(* IEC 61131-3 sources: AXOpen/src/components.keyence.vision/ctrl/src/Axo_IV3 (part 2) *)

                IF inParent = NULL THEN
                    Messenger.Activate(UINT#1500,eAxoMessageCategory#Error);
                    Status.Error.Id := UINT#1500;
                    RETURN;
                END_IF;
                IF Config.HWIDs.HW_Device  = UINT#0 THEN
                    Messenger.Activate(UINT#1501,eAxoMessageCategory#Error);
                    Status.Error.Id := UINT#1501;
                    RETURN;
                END_IF;
                IF Config.HWIDs.HwID_CommandControl  = UINT#0 THEN
                    Messenger.Activate(UINT#1502,eAxoMessageCategory#Error);
                    Status.Error.Id := UINT#1502;
                    RETURN;
                END_IF;
                IF Config.HWIDs.HwID_CommandStatusBits  = UINT#0 THEN
                    Messenger.Activate(UINT#1503,eAxoMessageCategory#Error);
                    Status.Error.Id := UINT#1503;
                    RETURN;
                END_IF;
                IF Config.HWIDs.HwID_DeviceResultBits_1  = UINT#0 THEN
                    Messenger.Activate(UINT#1504,eAxoMessageCategory#Error);
                    Status.Error.Id := UINT#1504;
                    RETURN;
                END_IF;
                IF Config.HWIDs.HwID_DeviceStatusWords  = UINT#0 THEN
                    Messenger.Activate(UINT#1505,eAxoMessageCategory#Error);
                    Status.Error.Id := UINT#1505;
                    RETURN;
                END_IF;
                IF Config.HWIDs.HwID_DeviceStatistics  = UINT#0 THEN
                    Messenger.Activate(UINT#1506,eAxoMessageCategory#Error);
                    Status.Error.Id := UINT#1506;
                    RETURN;
                END_IF;
                IF Config.HWIDs.HwID_PositionAdjustResult  = UINT#0 THEN
                    Messenger.Activate(UINT#1507,eAxoMessageCategory#Error);
                    Status.Error.Id := UINT#1507;
                    RETURN;
                END_IF;
                IF Config.HWIDs.HwID_ToolResult_1  = UINT#0 THEN
                    Messenger.Activate(UINT#1508,eAxoMessageCategory#Error);
                    Status.Error.Id := UINT#1508;
                    RETURN;
                END_IF;
                IF Config.HWIDs.HwID_ToolResult_2  = UINT#0 THEN
                    Messenger.Activate(UINT#1509,eAxoMessageCategory#Error);
                    Status.Error.Id := UINT#1509;
                    RETURN;
                END_IF;
                IF Config.HWIDs.HwID_ToolResult_3  = UINT#0 THEN
                    Messenger.Activate(UINT#1510,eAxoMessageCategory#Error);
                    Status.Error.Id := UINT#1510;
                    RETURN;
                END_IF;
                IF Config.HWIDs.HwID_ToolResult_4  = UINT#0 THEN
                    Messenger.Activate(UINT#1511,eAxoMessageCategory#Error);
                    Status.Error.Id := UINT#1511;
                    RETURN;
                END_IF;
                IF Config.HWIDs.HwID_ToolResult_5  = UINT#0 THEN
                    Messenger.Activate(UINT#1512,eAxoMessageCategory#Error);
                    Status.Error.Id := UINT#1512;
                    RETURN;
                END_IF;
                IF Config.HWIDs.HwID_ToolResult_6  = UINT#0 THEN
                    Messenger.Activate(UINT#1513,eAxoMessageCategory#Error);
                    Status.Error.Id := UINT#1513;
                    RETURN;
                END_IF;
                IF Config.HWIDs.HwID_ToolResult_7  = UINT#0 THEN
                    Messenger.Activate(UINT#1514,eAxoMessageCategory#Error);
                    Status.Error.Id := UINT#1514;
                    RETURN;
                END_IF;
                IF Config.HWIDs.HwID_ToolResult_8  = UINT#0 THEN
                    Messenger.Activate(UINT#1515,eAxoMessageCategory#Error);
                    Status.Error.Id := UINT#1515;
                    RETURN;
                END_IF;
                IF Config.HWIDs.HwID_ToolResult_9  = UINT#0 THEN
                    Messenger.Activate(UINT#1516,eAxoMessageCategory#Error);
                    Status.Error.Id := UINT#1516;
                    RETURN;
                END_IF;
                IF Config.HWIDs.HwID_ToolResult_10  = UINT#0 THEN
                    Messenger.Activate(UINT#1517,eAxoMessageCategory#Error);
                    Status.Error.Id := UINT#1517;
                    RETURN;
                END_IF;
                IF Config.HWIDs.HwID_ToolResult_11  = UINT#0 THEN
                    Messenger.Activate(UINT#1518,eAxoMessageCategory#Error);
                    Status.Error.Id := UINT#1518;
                    RETURN;
                END_IF;
                IF Config.HWIDs.HwID_ToolResult_12  = UINT#0 THEN
                    Messenger.Activate(UINT#1519,eAxoMessageCategory#Error);
                    Status.Error.Id := UINT#1519;
                    RETURN;
                END_IF;
                IF Config.HWIDs.HwID_ToolResult_13  = UINT#0 THEN
                    Messenger.Activate(UINT#1520,eAxoMessageCategory#Error);
                    Status.Error.Id := UINT#1520;
                    RETURN;
                END_IF;
                IF Config.HWIDs.HwID_ToolResult_14  = UINT#0 THEN
                    Messenger.Activate(UINT#1521,eAxoMessageCategory#Error);
                    Status.Error.Id := UINT#1521;
                    RETURN;
                END_IF;
                IF Config.HWIDs.HwID_ToolResult_15  = UINT#0 THEN
                    Messenger.Activate(UINT#1522,eAxoMessageCategory#Error);
                    Status.Error.Id := UINT#1522;
                    RETURN;
                END_IF;
                IF Config.HWIDs.HwID_ToolResult_16  = UINT#0 THEN
                    Messenger.Activate(UINT#1523,eAxoMessageCategory#Error);
                    Status.Error.Id := UINT#1523;
                    RETURN;
                END_IF;
                IF Config.HWIDs.HwID_ToolResult_17  = UINT#0 THEN
                    Messenger.Activate(UINT#1524,eAxoMessageCategory#Error);
                    Status.Error.Id := UINT#1524;
                    RETURN;
                END_IF;
                IF Config.HWIDs.HwID_ToolResult_18  = UINT#0 THEN
                    Messenger.Activate(UINT#1525,eAxoMessageCategory#Error);
                    Status.Error.Id := UINT#1525;
                    RETURN;
                END_IF;
                IF Config.HWIDs.HwID_ToolResult_19  = UINT#0 THEN
                    Messenger.Activate(UINT#1526,eAxoMessageCategory#Error);
                    Status.Error.Id := UINT#1526;
                    RETURN;
                END_IF;
                IF Config.HWIDs.HwID_ToolResult_20  = UINT#0 THEN
                    Messenger.Activate(UINT#1527,eAxoMessageCategory#Error);
                    Status.Error.Id := UINT#1527;
                    RETURN;
                END_IF;
                IF Config.HWIDs.HwID_ToolResult_21  = UINT#0 THEN
                    Messenger.Activate(UINT#1528,eAxoMessageCategory#Error);
                    Status.Error.Id := UINT#1528;
                    RETURN;
                END_IF;
                IF Config.HWIDs.HwID_ToolResult_22  = UINT#0 THEN
                    Messenger.Activate(UINT#1529,eAxoMessageCategory#Error);
                    Status.Error.Id := UINT#1529;
                    RETURN;
                END_IF;
                IF Config.HWIDs.HwID_ToolResult_23  = UINT#0 THEN
                    Messenger.Activate(UINT#1530,eAxoMessageCategory#Error);
                    Status.Error.Id := UINT#1530;
                    RETURN;
                END_IF;
                IF Config.HWIDs.HwID_ToolResult_24  = UINT#0 THEN
                    Messenger.Activate(UINT#1531,eAxoMessageCategory#Error);
                    Status.Error.Id := UINT#1531;
                    RETURN;
                END_IF;
                IF Config.HWIDs.HwID_ToolResult_25  = UINT#0 THEN
                    Messenger.Activate(UINT#1532,eAxoMessageCategory#Error);
                    Status.Error.Id := UINT#1532;
                    RETURN;
                END_IF;
                IF Config.HWIDs.HwID_ToolResult_26  = UINT#0 THEN
                    Messenger.Activate(UINT#1533,eAxoMessageCategory#Error);
                    Status.Error.Id := UINT#1533;
                    RETURN;
                END_IF;
                IF Config.HWIDs.HwID_ToolResult_27  = UINT#0 THEN
                    Messenger.Activate(UINT#1534,eAxoMessageCategory#Error);
                    Status.Error.Id := UINT#1534;
                    RETURN;
                END_IF;
                IF Config.HWIDs.HwID_ToolResult_28  = UINT#0 THEN
                    Messenger.Activate(UINT#1535,eAxoMessageCategory#Error);
                    Status.Error.Id := UINT#1535;
                    RETURN;
                END_IF;
                IF Config.HWIDs.HwID_ToolResult_29  = UINT#0 THEN
                    Messenger.Activate(UINT#1536,eAxoMessageCategory#Error);
                    Status.Error.Id := UINT#1536;
                    RETURN;
                END_IF;
                IF Config.HWIDs.HwID_ToolResult_30  = UINT#0 THEN
                    Messenger.Activate(UINT#1537,eAxoMessageCategory#Error);
                    Status.Error.Id := UINT#1537;
                    RETURN;
                END_IF;
                IF Config.HWIDs.HwID_ToolResult_31  = UINT#0 THEN
                    Messenger.Activate(UINT#1538,eAxoMessageCategory#Error);
                    Status.Error.Id := UINT#1538;
                    RETURN;
                END_IF;
                IF Config.HWIDs.HwID_ToolResult_32  = UINT#0 THEN
                    Messenger.Activate(UINT#1539,eAxoMessageCategory#Error);
                    Status.Error.Id := UINT#1539;
                    RETURN;
                END_IF;
                IF Config.HWIDs.HwID_ToolResult_33  = UINT#0 THEN
                    Messenger.Activate(UINT#1540,eAxoMessageCategory#Error);
                    Status.Error.Id := UINT#1540;
                    RETURN;
                END_IF;
                IF Config.HWIDs.HwID_ToolResult_34  = UINT#0 THEN
                    Messenger.Activate(UINT#1541,eAxoMessageCategory#Error);
                    Status.Error.Id := UINT#1541;
                    RETURN;
                END_IF;
                IF Config.HWIDs.HwID_ToolResult_35  = UINT#0 THEN
                    Messenger.Activate(UINT#1542,eAxoMessageCategory#Error);
                    Status.Error.Id := UINT#1542;
                    RETURN;
                END_IF;
                IF Config.HWIDs.HwID_ToolResult_36  = UINT#0 THEN
                    Messenger.Activate(UINT#1543,eAxoMessageCategory#Error);
                    Status.Error.Id := UINT#1543;
                    RETURN;
                END_IF;
                IF Config.HWIDs.HwID_ToolResult_37  = UINT#0 THEN
                    Messenger.Activate(UINT#1544,eAxoMessageCategory#Error);
                    Status.Error.Id := UINT#1544;
                    RETURN;
                END_IF;
                IF Config.HWIDs.HwID_ToolResult_38  = UINT#0 THEN
                    Messenger.Activate(UINT#1545,eAxoMessageCategory#Error);
                    Status.Error.Id := UINT#1545;
                    RETURN;
                END_IF;
                IF Config.HWIDs.HwID_ToolResult_39  = UINT#0 THEN
                    Messenger.Activate(UINT#1546,eAxoMessageCategory#Error);
                    Status.Error.Id := UINT#1546;
                    RETURN;
                END_IF;
                IF Config.HWIDs.HwID_ToolResult_40  = UINT#0 THEN
                    Messenger.Activate(UINT#1547,eAxoMessageCategory#Error);
                    Status.Error.Id := UINT#1547;
                    RETURN;
                END_IF;
                IF Config.HWIDs.HwID_ToolResult_41  = UINT#0 THEN
                    Messenger.Activate(UINT#1548,eAxoMessageCategory#Error);
                    Status.Error.Id := UINT#1548;
                    RETURN;
                END_IF;
                IF Config.HWIDs.HwID_ToolResult_42  = UINT#0 THEN
                    Messenger.Activate(UINT#1549,eAxoMessageCategory#Error);
                    Status.Error.Id := UINT#1549;
                    RETURN;
                END_IF;
                IF Config.HWIDs.HwID_ToolResult_43  = UINT#0 THEN
                    Messenger.Activate(UINT#1550,eAxoMessageCategory#Error);
                    Status.Error.Id := UINT#1550;
                    RETURN;
                END_IF;
                IF Config.HWIDs.HwID_ToolResult_44  = UINT#0 THEN
                    Messenger.Activate(UINT#1551,eAxoMessageCategory#Error);
                    Status.Error.Id := UINT#1551;
                    RETURN;
                END_IF;
                IF Config.HWIDs.HwID_ToolResult_45  = UINT#0 THEN
                    Messenger.Activate(UINT#1552,eAxoMessageCategory#Error);
                    Status.Error.Id := UINT#1552;
                    RETURN;
                END_IF;
                IF Config.HWIDs.HwID_ToolResult_46  = UINT#0 THEN
                    Messenger.Activate(UINT#1553,eAxoMessageCategory#Error);
                    Status.Error.Id := UINT#1553;
                    RETURN;
                END_IF;
                IF Config.HWIDs.HwID_ToolResult_47  = UINT#0 THEN
                    Messenger.Activate(UINT#1554,eAxoMessageCategory#Error);
                    Status.Error.Id := UINT#1554;
                    RETURN;
                END_IF;
                IF Config.HWIDs.HwID_ToolResult_48  = UINT#0 THEN
                    Messenger.Activate(UINT#1555,eAxoMessageCategory#Error);
                    Status.Error.Id := UINT#1555;
                    RETURN;
                END_IF;
                IF Config.HWIDs.HwID_ToolResult_49  = UINT#0 THEN
                    Messenger.Activate(UINT#1556,eAxoMessageCategory#Error);
                    Status.Error.Id := UINT#1556;
                    RETURN;
                END_IF;
                IF Config.HWIDs.HwID_ToolResult_50  = UINT#0 THEN
                    Messenger.Activate(UINT#1557,eAxoMessageCategory#Error);
                    Status.Error.Id := UINT#1557;
                    RETURN;
                END_IF;
                IF Config.HWIDs.HwID_ToolResult_51  = UINT#0 THEN
                    Messenger.Activate(UINT#1558,eAxoMessageCategory#Error);
                    Status.Error.Id := UINT#1558;
                    RETURN;
                END_IF;
                IF Config.HWIDs.HwID_ToolResult_52  = UINT#0 THEN
                    Messenger.Activate(UINT#1559,eAxoMessageCategory#Error);
                    Status.Error.Id := UINT#1559;
                    RETURN;
                END_IF;
                IF Config.HWIDs.HwID_ToolResult_53  = UINT#0 THEN
                    Messenger.Activate(UINT#1560,eAxoMessageCategory#Error);
                    Status.Error.Id := UINT#1560;
                    RETURN;
                END_IF;
                IF Config.HWIDs.HwID_ToolResult_54  = UINT#0 THEN
                    Messenger.Activate(UINT#1561,eAxoMessageCategory#Error);
                    Status.Error.Id := UINT#1561;
                    RETURN;
                END_IF;
                IF Config.HWIDs.HwID_ToolResult_55  = UINT#0 THEN
                    Messenger.Activate(UINT#1562,eAxoMessageCategory#Error);
                    Status.Error.Id := UINT#1562;
                    RETURN;
                END_IF;
                IF Config.HWIDs.HwID_ToolResult_56  = UINT#0 THEN
                    Messenger.Activate(UINT#1563,eAxoMessageCategory#Error);
                    Status.Error.Id := UINT#1563;
                    RETURN;
                END_IF;
                IF Config.HWIDs.HwID_ToolResult_57  = UINT#0 THEN
                    Messenger.Activate(UINT#1564,eAxoMessageCategory#Error);
                    Status.Error.Id := UINT#1564;
                    RETURN;
                END_IF;
                IF Config.HWIDs.HwID_ToolResult_58  = UINT#0 THEN
                    Messenger.Activate(UINT#1565,eAxoMessageCategory#Error);
                    Status.Error.Id := UINT#1565;
                    RETURN;
                END_IF;
                IF Config.HWIDs.HwID_ToolResult_59  = UINT#0 THEN
                    Messenger.Activate(UINT#1566,eAxoMessageCategory#Error);
                    Status.Error.Id := UINT#1566;
                    RETURN;
                END_IF;
                IF Config.HWIDs.HwID_ToolResult_60  = UINT#0 THEN
                    Messenger.Activate(UINT#1567,eAxoMessageCategory#Error);
                    Status.Error.Id := UINT#1567;
                    RETURN;
                END_IF;
                IF Config.HWIDs.HwID_ToolResult_61  = UINT#0 THEN
                    Messenger.Activate(UINT#1568,eAxoMessageCategory#Error);
                    Status.Error.Id := UINT#1568;
                    RETURN;
                END_IF;
                IF Config.HWIDs.HwID_ToolResult_62  = UINT#0 THEN
                    Messenger.Activate(UINT#1569,eAxoMessageCategory#Error);
                    Status.Error.Id := UINT#1569;
                    RETURN;
                END_IF;
                IF Config.HWIDs.HwID_ToolResult_63  = UINT#0 THEN
                    Messenger.Activate(UINT#1570,eAxoMessageCategory#Error);
                    Status.Error.Id := UINT#1570;
                    RETURN;
                END_IF;
                IF Config.HWIDs.HwID_ToolResult_64  = UINT#0 THEN
                    Messenger.Activate(UINT#1571,eAxoMessageCategory#Error);
                    Status.Error.Id := UINT#1571;
                    RETURN;
                END_IF;
                IF Config.HWIDs.HwID_DeviceResultBits_2  = UINT#0 THEN
                    Messenger.Activate(UINT#1572,eAxoMessageCategory#Error);
                    Status.Error.Id := UINT#1572;
                    RETURN;
                END_IF;

                _initHwCheckDone    := TRUE;
            END_IF;

            //***********Update inputs **************
            //*************************CommandStatusBits*********************
            _retVal := Siemens.Simatic.DistributedIO.ReadData((Config.HWIDs.HwID_CommandStatusBits) ,_data_in);
            IF _retVal > WORD#0 THEN
                Messenger.Activate(UINT#1601, eAxoMessageCategory#Error);
                Status.Error.Id := UINT#1601;
                RETURN;
            END_IF;

            Inputs.CommandStatusBits.TriggerResponse               :=   _data_in[0].%X0;       // IB0.0
            Inputs.CommandStatusBits.MasterRegistrationResponse    :=   _data_in[0].%X1;       // IB0.1
            Inputs.CommandStatusBits.ProgramSwitchingResponse      :=   _data_in[0].%X2;       // IB0.2
            Inputs.CommandStatusBits.WarningClearResponse          :=   _data_in[0].%X3;       // IB0.3
            Inputs.CommandStatusBits.StatisticsResetResponse       :=   _data_in[0].%X4;       // IB0.4
            Inputs.CommandStatusBits.BufferClearResponse           :=   _data_in[0].%X5;       // IB0.5
            Inputs.CommandStatusBits.SdCardSavingStopResponse      :=   _data_in[0].%X6;       // IB0.6
            Inputs.CommandStatusBits.SettingValueChangeResponse    :=   _data_in[0].%X7;       // IB0.7

            Inputs.CommandStatusBits.TriggerFailed                 :=   _data_in[1].%X0;       // IB1.0
            Inputs.CommandStatusBits.MasterRegistrationFailed      :=   _data_in[1].%X1;       // IB1.1
            Inputs.CommandStatusBits.ProgramSwitchingFailed        :=   _data_in[1].%X2;       // IB1.2
                                                               //  :=   _data_in[1].%X3;       // IB1.3
                                                               //  :=   _data_in[1].%X4;       // IB1.4
                                                               //  :=   _data_in[1].%X5;       // IB1.5
            Inputs.CommandStatusBits.SdCardSavingStopFailed        :=   _data_in[1].%X6;       // IB1.6
            Inputs.CommandStatusBits.SettingValueChangeFailed      :=   _data_in[1].%X7;       // IB1.7

            Inputs.CommandStatusBits.ResultAvailable               :=   _data_in[2].%X0;       // IB2.0
            Inputs.CommandStatusBits.ResultUpdateComplete          :=   _data_in[2].%X1;       // IB2.1
            Inputs.CommandStatusBits.BUSY                          :=   _data_in[2].%X2;       // IB2.2
            Inputs.CommandStatusBits.ImagingStatus                 :=   _data_in[2].%X3;       // IB2.3
            Inputs.CommandStatusBits.RUN                           :=   _data_in[2].%X4;       // IB2.4
            Inputs.CommandStatusBits.Ready                         :=   _data_in[2].%X5;       // IB2.5
            Inputs.CommandStatusBits.TriggerReady                  :=   _data_in[2].%X6;       // IB2.6
            Inputs.CommandStatusBits.SdCardIdentificationStatus    :=   _data_in[2].%X7;       // IB2.7

            Inputs.CommandStatusBits.SortingModeInformation        :=   _data_in[3].%X0;       // IB3.0
                                                                // :=   _data_in[3].%X1;       // IB3.1
                                                                // :=   _data_in[3].%X2;       // IB3.2
                                                                // :=   _data_in[3].%X3;       // IB3.3
            Inputs.CommandStatusBits.InsufficientFreeSpaceOnSdCard :=   _data_in[3].%X4;       // IB3.4
            Inputs.CommandStatusBits.BufferOverrun                 :=   _data_in[3].%X5;       // IB3.5
            Inputs.CommandStatusBits.Warning                       :=   _data_in[3].%X6;       // IB3.6
            Inputs.CommandStatusBits.Error                         :=   _data_in[3].%X7;       // IB3.7
            //***************************************************************

            //*************************DeviceResultBits_1********************
            _retVal := Siemens.Simatic.DistributedIO.ReadData((Config.HWIDs.HwID_DeviceResultBits_1) ,_data_in);
            IF _retVal > WORD#0 THEN
                Messenger.Activate(UINT#1602, eAxoMessageCategory#Error);
                Status.Error.Id := UINT#1602;
                RETURN;
            END_IF;

            Inputs.DeviceResultBits_1.OverallJudgmentOK             :=   _data_in[0].%X0;       // IB4.0
            Inputs.DeviceResultBits_1.PositionCorrection            :=   _data_in[0].%X1;       // IB4.1
            Inputs.DeviceResultBits_1.LOGIC1                        :=   _data_in[0].%X2;       // IB4.2
            Inputs.DeviceResultBits_1.LOGIC2                        :=   _data_in[0].%X3;       // IB4.3
            Inputs.DeviceResultBits_1.LOGIC3                        :=   _data_in[0].%X4;       // IB4.4
            Inputs.DeviceResultBits_1.LOGIC4                        :=   _data_in[0].%X5;       // IB4.5
            Inputs.DeviceResultBits_1.OverallJudgmentNG             :=   _data_in[0].%X6;       // IB4.6
                                                                 // :=   _data_in[0].%X7;       // IB4.7

            Inputs.DeviceResultBits_1.Tool_1                        :=   _data_in[2].%X0;       // IB6.0
            Inputs.DeviceResultBits_1.Tool_2                        :=   _data_in[2].%X1;       // IB6.1
            Inputs.DeviceResultBits_1.Tool_3                        :=   _data_in[2].%X2;       // IB6.2
            Inputs.DeviceResultBits_1.Tool_4                        :=   _data_in[2].%X3;       // IB6.3
            Inputs.DeviceResultBits_1.Tool_5                        :=   _data_in[2].%X4;       // IB6.4
            Inputs.DeviceResultBits_1.Tool_6                        :=   _data_in[2].%X5;       // IB6.5
            Inputs.DeviceResultBits_1.Tool_7                        :=   _data_in[2].%X6;       // IB6.6
            Inputs.DeviceResultBits_1.Tool_8                        :=   _data_in[2].%X7;       // IB6.7

            Inputs.DeviceResultBits_1.Tool_9                        :=   _data_in[3].%X0;       // IB7.0
            Inputs.DeviceResultBits_1.Tool_10                       :=   _data_in[3].%X1;       // IB7.1
            Inputs.DeviceResultBits_1.Tool_11                       :=   _data_in[3].%X2;       // IB7.2
            Inputs.DeviceResultBits_1.Tool_12                       :=   _data_in[3].%X3;       // IB7.3
            Inputs.DeviceResultBits_1.Tool_13                       :=   _data_in[3].%X4;       // IB7.4
            Inputs.DeviceResultBits_1.Tool_14                       :=   _data_in[3].%X5;       // IB7.5
            Inputs.DeviceResultBits_1.Tool_15                       :=   _data_in[3].%X6;       // IB7.6
            Inputs.DeviceResultBits_1.Tool_16                       :=   _data_in[3].%X7;       // IB7.7
            //***************************************************************

            //*************************DeviceStatusWords*********************
            _retVal := Siemens.Simatic.DistributedIO.ReadData((Config.HWIDs.HwID_DeviceStatusWords) ,_data_in);
            IF _retVal > WORD#0 THEN
                Messenger.Activate(UINT#1603, eAxoMessageCategory#Error);
                Status.Error.Id := UINT#1603;
                RETURN;
            END_IF;

            _word.%B0 := _data_in[1];
            _word.%B1 := _data_in[0];
            Inputs.DeviceStatusWords.ErrorNo                       :=  TO_UINT(_word);         // IW8
            _word.%B0 := _data_in[3];
            _word.%B1 := _data_in[2];
            Inputs.DeviceStatusWords.WarningNo                     :=  TO_UINT(_word);         // IW10
            _word.%B0 := _data_in[5];
            _word.%B1 := _data_in[4];
            Inputs.DeviceStatusWords.NumberOfRemainingBuffers      :=  TO_UINT(_word);         // IW12
            _word.%B0 := _data_in[7];
            _word.%B1 := _data_in[6];
            Inputs.DeviceStatusWords.Checksum                      :=  TO_UINT(_word);         // IW14
            _word.%B0 := _data_in[9];
            _word.%B1 := _data_in[8];
            Inputs.DeviceStatusWords.CurrentProgramNo              :=  TO_UINT(_word);         // IW16
            _word.%B0 := _data_in[11];
            _word.%B1 := _data_in[10];
            Inputs.DeviceStatusWords.ProgramNoDuringJudgment       :=  TO_UINT(_word);         // IW18
            _word.%B0 := _data_in[13];
            _word.%B1 := _data_in[12];
            Inputs.DeviceStatusWords.ResultNo                      :=  TO_UINT(_word);         // IW20
            _word.%B0 := _data_in[15];
            _word.%B1 := _data_in[14];
            Inputs.DeviceStatusWords.ProcessingTime                :=  TO_UINT(_word);         // IW22
            //***************************************************************

            //*************************DeviceStatistics**********************
            _retVal := Siemens.Simatic.DistributedIO.ReadData((Config.HWIDs.HwID_DeviceStatistics) ,_data_in);
            IF _retVal > WORD#0 THEN
                Messenger.Activate(UINT#1604, eAxoMessageCategory#Error);
                Status.Error.Id := UINT#1604;
                RETURN;
            END_IF;

            _word.%B0 := _data_in[1];
            _word.%B1 := _data_in[0];
            Inputs.DeviceStatistics.ProcessingTimeMax             :=  TO_UINT(_word);         // IW24
            _word.%B0 := _data_in[3];
            _word.%B1 := _data_in[2];
            Inputs.DeviceStatistics.ProcessingTimeMin             :=  TO_UINT(_word);         // IW26
            _word.%B0 := _data_in[5];
            _word.%B1 := _data_in[4];
            Inputs.DeviceStatistics.ProcessingTimeAve             :=  TO_UINT(_word);         // IW28
                                                                                              // IW30
            _dword.%B0 := _data_in[11];
            _dword.%B1 := _data_in[10];
            _dword.%B2 := _data_in[9];
            _dword.%B3 := _data_in[8];
            Inputs.DeviceStatistics.NumberOfTriggers              :=  TO_UINT(_dword);        // ID32
            _dword.%B0 := _data_in[15];
            _dword.%B1 := _data_in[14];
            _dword.%B2 := _data_in[13];
            _dword.%B3 := _data_in[12];
            Inputs.DeviceStatistics.NumberOfOKs                   :=  TO_UINT(_dword);        // ID36
            _dword.%B0 := _data_in[19];
            _dword.%B1 := _data_in[18];
            _dword.%B2 := _data_in[17];
            _dword.%B3 := _data_in[16];
            Inputs.DeviceStatistics.NumberOfNGs                   :=  TO_UINT(_dword);        // ID40
            _dword.%B0 := _data_in[23];
            _dword.%B1 := _data_in[22];
            _dword.%B2 := _data_in[21];
            _dword.%B3 := _data_in[20];
            Inputs.DeviceStatistics.NumberOfTriggerErrors         :=  TO_UINT(_dword);        // ID44
                                                                                              // ID48
            //***************************************************************

            //*************************PositionAdjustResult******************
            _retVal := Siemens.Simatic.DistributedIO.ReadData((Config.HWIDs.HwID_PositionAdjustResult) ,_data_in);
            IF _retVal > WORD#0 THEN
                Messenger.Activate(UINT#1605, eAxoMessageCategory#Error);
                Status.Error.Id := UINT#1605;
                RETURN;
            END_IF;

            _word.%B0 := _data_in[1];
            _word.%B1 := _data_in[0];
            Inputs.PositionAdjustResult.PositionCorrectionScore       :=  TO_UINT(_word);         // IW52
            _word.%B0 := _data_in[3];
            _word.%B1 := _data_in[2];
            Inputs.PositionAdjustResult.PositionCorrectionScoreMAX    :=  TO_UINT(_word);         // IW54
            _word.%B0 := _data_in[5];
            _word.%B1 := _data_in[4];
            Inputs.PositionAdjustResult.PositionCorrectionScoreMIN    :=  TO_UINT(_word);         // IW56
            _word.%B0 := _data_in[7];
            _word.%B1 := _data_in[6];
            Inputs.PositionAdjustResult.PositionCorrectionScoreLowerThreshold :=  TO_UINT(_word); // IW58
                                                                                                  // IB60-IB71
            //***************************************************************

            //*************************ToolResult_1**************************
            _retVal := Siemens.Simatic.DistributedIO.ReadData((Config.HWIDs.HwID_ToolResult_1) ,_data_in);
            IF _retVal > WORD#0 THEN
                Messenger.Activate(UINT#1606, eAxoMessageCategory#Error);
                Status.Error.Id := UINT#1606;
                RETURN;
            END_IF;

            _word.%B0 := _data_in[1];
            _word.%B1 := _data_in[0];
            Inputs.ToolResult_1.MatchingRate       :=  TO_UINT(_word);         // IW72
            _word.%B0 := _data_in[3];
            _word.%B1 := _data_in[2];
            Inputs.ToolResult_1.MatchingRateMAX    :=  TO_UINT(_word);         // IW74
            _word.%B0 := _data_in[5];
            _word.%B1 := _data_in[4];
            Inputs.ToolResult_1.MatchingRateMIN    :=  TO_UINT(_word);         // IW76
            _word.%B0 := _data_in[7];
            _word.%B1 := _data_in[6];
            Inputs.ToolResult_1.LowerThreshold     :=  TO_UINT(_word);         // IW78
            _word.%B0 := _data_in[9];
            _word.%B1 := _data_in[8];
            Inputs.ToolResult_1.UpperThreshold     :=  TO_UINT(_word);         // IW80
            _word.%B0 := _data_in[11];
            _word.%B1 := _data_in[10];
            Inputs.ToolResult_1.DecimalPointPosition:=  TO_UINT(_word);        // IW82
            _word.%B0 := _data_in[13];
            _word.%B1 := _data_in[12];
            Inputs.ToolResult_1.Data_1             :=  TO_UINT(_word);         // IW84
            _word.%B0 := _data_in[15];
            _word.%B1 := _data_in[14];
            Inputs.ToolResult_1.Data_2             :=  TO_UINT(_word);         // IW86
            _word.%B0 := _data_in[17];
            _word.%B1 := _data_in[16];
            Inputs.ToolResult_1.Data_3             :=  TO_UINT(_word);         // IW88
                                                                                    // IW90
            //***************************************************************

            //*************************ToolResult_2**************************
            _retVal := Siemens.Simatic.DistributedIO.ReadData((Config.HWIDs.HwID_ToolResult_2) ,_data_in);
            IF _retVal > WORD#0 THEN
                Messenger.Activate(UINT#1607, eAxoMessageCategory#Error);
                Status.Error.Id := UINT#1607;
                RETURN;
            END_IF;

            _word.%B0 := _data_in[1];
            _word.%B1 := _data_in[0];
            Inputs.ToolResult_2.MatchingRate       :=  TO_UINT(_word);         // IW92
            _word.%B0 := _data_in[3];
            _word.%B1 := _data_in[2];
            Inputs.ToolResult_2.MatchingRateMAX    :=  TO_UINT(_word);         // IW94
            _word.%B0 := _data_in[5];
            _word.%B1 := _data_in[4];
            Inputs.ToolResult_2.MatchingRateMIN    :=  TO_UINT(_word);         // IW96
            _word.%B0 := _data_in[7];
            _word.%B1 := _data_in[6];
            Inputs.ToolResult_2.LowerThreshold     :=  TO_UINT(_word);         // IW98
            _word.%B0 := _data_in[9];
            _word.%B1 := _data_in[8];
            Inputs.ToolResult_2.UpperThreshold     :=  TO_UINT(_word);         // IW100
            _word.%B0 := _data_in[11];
            _word.%B1 := _data_in[10];
            Inputs.ToolResult_2.DecimalPointPosition:=  TO_UINT(_word);        // IW102
            _word.%B0 := _data_in[13];
            _word.%B1 := _data_in[12];
            Inputs.ToolResult_2.Data_1             :=  TO_UINT(_word);         // IW104
            _word.%B0 := _data_in[15];
            _word.%B1 := _data_in[14];
            Inputs.ToolResult_2.Data_2             :=  TO_UINT(_word);         // IW106
            _word.%B0 := _data_in[17];
            _word.%B1 := _data_in[16];
            Inputs.ToolResult_2.Data_3             :=  TO_UINT(_word);         // IW108
                                                                                    // IW110
            //***************************************************************

            //*************************ToolResult_3**************************
            _retVal := Siemens.Simatic.DistributedIO.ReadData((Config.HWIDs.HwID_ToolResult_3) ,_data_in);
            IF _retVal > WORD#0 THEN
                Messenger.Activate(UINT#1608, eAxoMessageCategory#Error);
                Status.Error.Id := UINT#1608;
                RETURN;
            END_IF;

            _word.%B0 := _data_in[1];
            _word.%B1 := _data_in[0];
            Inputs.ToolResult_3.MatchingRate       :=  TO_UINT(_word);         // IW112
            _word.%B0 := _data_in[3];
            _word.%B1 := _data_in[2];
            Inputs.ToolResult_3.MatchingRateMAX    :=  TO_UINT(_word);         // IW114
            _word.%B0 := _data_in[5];
            _word.%B1 := _data_in[4];
            Inputs.ToolResult_3.MatchingRateMIN    :=  TO_UINT(_word);         // IW116
            _word.%B0 := _data_in[7];
            _word.%B1 := _data_in[6];
            Inputs.ToolResult_3.LowerThreshold     :=  TO_UINT(_word);         // IW118
            _word.%B0 := _data_in[9];
            _word.%B1 := _data_in[8];
            Inputs.ToolResult_3.UpperThreshold     :=  TO_UINT(_word);         // IW120
            _word.%B0 := _data_in[11];
            _word.%B1 := _data_in[10];
            Inputs.ToolResult_3.DecimalPointPosition:=  TO_UINT(_word);        // IW122
            _word.%B0 := _data_in[13];
            _word.%B1 := _data_in[12];
            Inputs.ToolResult_3.Data_1             :=  TO_UINT(_word);         // IW124
            _word.%B0 := _data_in[15];
            _word.%B1 := _data_in[14];
            Inputs.ToolResult_3.Data_2             :=  TO_UINT(_word);         // IW126
            _word.%B0 := _data_in[17];
            _word.%B1 := _data_in[16];
            Inputs.ToolResult_3.Data_3             :=  TO_UINT(_word);         // IW128
                                                                                    // IW130
            //***************************************************************

            //*************************ToolResult_4**************************
            _retVal := Siemens.Simatic.DistributedIO.ReadData((Config.HWIDs.HwID_ToolResult_4) ,_data_in);
            IF _retVal > WORD#0 THEN
                Messenger.Activate(UINT#1609, eAxoMessageCategory#Error);
                Status.Error.Id := UINT#1609;
                RETURN;
            END_IF;

            _word.%B0 := _data_in[1];
            _word.%B1 := _data_in[0];
            Inputs.ToolResult_4.MatchingRate       :=  TO_UINT(_word);         // IW132
            _word.%B0 := _data_in[3];
            _word.%B1 := _data_in[2];
            Inputs.ToolResult_4.MatchingRateMAX    :=  TO_UINT(_word);         // IW134
            _word.%B0 := _data_in[5];
            _word.%B1 := _data_in[4];
            Inputs.ToolResult_4.MatchingRateMIN    :=  TO_UINT(_word);         // IW136
            _word.%B0 := _data_in[7];
            _word.%B1 := _data_in[6];
            Inputs.ToolResult_4.LowerThreshold     :=  TO_UINT(_word);         // IW138
            _word.%B0 := _data_in[9];
            _word.%B1 := _data_in[8];
            Inputs.ToolResult_4.UpperThreshold     :=  TO_UINT(_word);         // IW140
            _word.%B0 := _data_in[11];
            _word.%B1 := _data_in[10];
            Inputs.ToolResult_4.DecimalPointPosition:=  TO_UINT(_word);        // IW142
            _word.%B0 := _data_in[13];
            _word.%B1 := _data_in[12];
            Inputs.ToolResult_4.Data_1             :=  TO_UINT(_word);         // IW144
            _word.%B0 := _data_in[15];
            _word.%B1 := _data_in[14];
            Inputs.ToolResult_4.Data_2             :=  TO_UINT(_word);         // IW146
            _word.%B0 := _data_in[17];
            _word.%B1 := _data_in[16];
            Inputs.ToolResult_4.Data_3             :=  TO_UINT(_word);         // IW148
                                                                                    // IW150
            //***************************************************************

            //*************************ToolResult_5**************************
            _retVal := Siemens.Simatic.DistributedIO.ReadData((Config.HWIDs.HwID_ToolResult_5) ,_data_in);
            IF _retVal > WORD#0 THEN
                Messenger.Activate(UINT#1610, eAxoMessageCategory#Error);
                Status.Error.Id := UINT#1610;
                RETURN;
            END_IF;

            _word.%B0 := _data_in[1];
            _word.%B1 := _data_in[0];
            Inputs.ToolResult_5.MatchingRate       :=  TO_UINT(_word);         // IW152
            _word.%B0 := _data_in[3];
            _word.%B1 := _data_in[2];
            Inputs.ToolResult_5.MatchingRateMAX    :=  TO_UINT(_word);         // IW154
            _word.%B0 := _data_in[5];
            _word.%B1 := _data_in[4];
            Inputs.ToolResult_5.MatchingRateMIN    :=  TO_UINT(_word);         // IW156
            _word.%B0 := _data_in[7];
            _word.%B1 := _data_in[6];
            Inputs.ToolResult_5.LowerThreshold     :=  TO_UINT(_word);         // IW158
            _word.%B0 := _data_in[9];
            _word.%B1 := _data_in[8];
            Inputs.ToolResult_5.UpperThreshold     :=  TO_UINT(_word);         // IW160
            _word.%B0 := _data_in[11];
            _word.%B1 := _data_in[10];
            Inputs.ToolResult_5.DecimalPointPosition:=  TO_UINT(_word);        // IW162
            _word.%B0 := _data_in[13];
            _word.%B1 := _data_in[12];
            Inputs.ToolResult_5.Data_1             :=  TO_UINT(_word);         // IW164
            _word.%B0 := _data_in[15];
            _word.%B1 := _data_in[14];
            Inputs.ToolResult_5.Data_2             :=  TO_UINT(_word);         // IW166
            _word.%B0 := _data_in[17];
            _word.%B1 := _data_in[16];
            Inputs.ToolResult_5.Data_3             :=  TO_UINT(_word);         // IW168
                                                                                    // IW170
            //***************************************************************

            //*************************ToolResult_6**************************
            _retVal := Siemens.Simatic.DistributedIO.ReadData((Config.HWIDs.HwID_ToolResult_6) ,_data_in);
            IF _retVal > WORD#0 THEN
                Messenger.Activate(UINT#1611, eAxoMessageCategory#Error);
                Status.Error.Id := UINT#1611;
                RETURN;
            END_IF;

            _word.%B0 := _data_in[1];
            _word.%B1 := _data_in[0];
            Inputs.ToolResult_6.MatchingRate       :=  TO_UINT(_word);         // IW172
            _word.%B0 := _data_in[3];
            _word.%B1 := _data_in[2];
            Inputs.ToolResult_6.MatchingRateMAX    :=  TO_UINT(_word);         // IW174
            _word.%B0 := _data_in[5];
            _word.%B1 := _data_in[4];
            Inputs.ToolResult_6.MatchingRateMIN    :=  TO_UINT(_word);         // IW176
            _word.%B0 := _data_in[7];
            _word.%B1 := _data_in[6];
            Inputs.ToolResult_6.LowerThreshold     :=  TO_UINT(_word);         // IW178
            _word.%B0 := _data_in[9];
            _word.%B1 := _data_in[8];
            Inputs.ToolResult_6.UpperThreshold     :=  TO_UINT(_word);         // IW180
            _word.%B0 := _data_in[11];
            _word.%B1 := _data_in[10];
            Inputs.ToolResult_6.DecimalPointPosition:=  TO_UINT(_word);        // IW182
            _word.%B0 := _data_in[13];
            _word.%B1 := _data_in[12];
            Inputs.ToolResult_6.Data_1             :=  TO_UINT(_word);         // IW184
            _word.%B0 := _data_in[15];
            _word.%B1 := _data_in[14];
            Inputs.ToolResult_6.Data_2             :=  TO_UINT(_word);         // IW186
            _word.%B0 := _data_in[17];
            _word.%B1 := _data_in[16];
            Inputs.ToolResult_6.Data_3             :=  TO_UINT(_word);         // IW188
                                                                                    // IW190
            //***************************************************************

            //*************************ToolResult_7**************************
            _retVal := Siemens.Simatic.DistributedIO.ReadData((Config.HWIDs.HwID_ToolResult_7) ,_data_in);
            IF _retVal > WORD#0 THEN
                Messenger.Activate(UINT#1612, eAxoMessageCategory#Error);
                Status.Error.Id := UINT#1612;
                RETURN;
            END_IF;

            _word.%B0 := _data_in[1];
            _word.%B1 := _data_in[0];
            Inputs.ToolResult_7.MatchingRate       :=  TO_UINT(_word);         // IW192
            _word.%B0 := _data_in[3];
            _word.%B1 := _data_in[2];
            Inputs.ToolResult_7.MatchingRateMAX    :=  TO_UINT(_word);         // IW194
            _word.%B0 := _data_in[5];
            _word.%B1 := _data_in[4];
            Inputs.ToolResult_7.MatchingRateMIN    :=  TO_UINT(_word);         // IW196
            _word.%B0 := _data_in[7];
            _word.%B1 := _data_in[6];
            Inputs.ToolResult_7.LowerThreshold     :=  TO_UINT(_word);         // IW198
            _word.%B0 := _data_in[9];
            _word.%B1 := _data_in[8];
            Inputs.ToolResult_7.UpperThreshold     :=  TO_UINT(_word);         // IW200
            _word.%B0 := _data_in[11];
            _word.%B1 := _data_in[10];
            Inputs.ToolResult_7.DecimalPointPosition:=  TO_UINT(_word);        // IW202
            _word.%B0 := _data_in[13];
            _word.%B1 := _data_in[12];
            Inputs.ToolResult_7.Data_1             :=  TO_UINT(_word);         // IW204
            _word.%B0 := _data_in[15];
            _word.%B1 := _data_in[14];
            Inputs.ToolResult_7.Data_2             :=  TO_UINT(_word);         // IW206
            _word.%B0 := _data_in[17];
            _word.%B1 := _data_in[16];
            Inputs.ToolResult_7.Data_3             :=  TO_UINT(_word);         // IW208
                                                                                    // IW210
            //***************************************************************

            //*************************ToolResult_8**************************
            _retVal := Siemens.Simatic.DistributedIO.ReadData((Config.HWIDs.HwID_ToolResult_8) ,_data_in);
            IF _retVal > WORD#0 THEN
                Messenger.Activate(UINT#1613, eAxoMessageCategory#Error);
                Status.Error.Id := UINT#1613;
                RETURN;
            END_IF;

            _word.%B0 := _data_in[1];
            _word.%B1 := _data_in[0];
            Inputs.ToolResult_8.MatchingRate       :=  TO_UINT(_word);         // IW212
            _word.%B0 := _data_in[3];
            _word.%B1 := _data_in[2];
            Inputs.ToolResult_8.MatchingRateMAX    :=  TO_UINT(_word);         // IW214
            _word.%B0 := _data_in[5];
            _word.%B1 := _data_in[4];
            Inputs.ToolResult_8.MatchingRateMIN    :=  TO_UINT(_word);         // IW216
            _word.%B0 := _data_in[7];
            _word.%B1 := _data_in[6];
            Inputs.ToolResult_8.LowerThreshold     :=  TO_UINT(_word);         // IW218
            _word.%B0 := _data_in[9];
            _word.%B1 := _data_in[8];
            Inputs.ToolResult_8.UpperThreshold     :=  TO_UINT(_word);         // IW220
            _word.%B0 := _data_in[11];
            _word.%B1 := _data_in[10];
            Inputs.ToolResult_8.DecimalPointPosition:=  TO_UINT(_word);        // IW222
            _word.%B0 := _data_in[13];
            _word.%B1 := _data_in[12];
            Inputs.ToolResult_8.Data_1             :=  TO_UINT(_word);         // IW224
            _word.%B0 := _data_in[15];
            _word.%B1 := _data_in[14];
            Inputs.ToolResult_8.Data_2             :=  TO_UINT(_word);         // IW226
            _word.%B0 := _data_in[17];
            _word.%B1 := _data_in[16];
            Inputs.ToolResult_8.Data_3             :=  TO_UINT(_word);         // IW228
                                                                                    // IW230
            //***************************************************************

            //*************************ToolResult_9**************************
            _retVal := Siemens.Simatic.DistributedIO.ReadData((Config.HWIDs.HwID_ToolResult_9) ,_data_in);
            IF _retVal > WORD#0 THEN
                Messenger.Activate(UINT#1614, eAxoMessageCategory#Error);
                Status.Error.Id := UINT#1614;
                RETURN;
            END_IF;

            _word.%B0 := _data_in[1];
            _word.%B1 := _data_in[0];
            Inputs.ToolResult_9.MatchingRate       :=  TO_UINT(_word);         // IW232
            _word.%B0 := _data_in[3];
            _word.%B1 := _data_in[2];
            Inputs.ToolResult_9.MatchingRateMAX    :=  TO_UINT(_word);         // IW234
            _word.%B0 := _data_in[5];
            _word.%B1 := _data_in[4];
            Inputs.ToolResult_9.MatchingRateMIN    :=  TO_UINT(_word);         // IW236
            _word.%B0 := _data_in[7];
            _word.%B1 := _data_in[6];
            Inputs.ToolResult_9.LowerThreshold     :=  TO_UINT(_word);         // IW238
            _word.%B0 := _data_in[9];
            _word.%B1 := _data_in[8];
            Inputs.ToolResult_9.UpperThreshold     :=  TO_UINT(_word);         // IW240
            _word.%B0 := _data_in[11];
            _word.%B1 := _data_in[10];
            Inputs.ToolResult_9.DecimalPointPosition:=  TO_UINT(_word);        // IW242
            _word.%B0 := _data_in[13];
            _word.%B1 := _data_in[12];
            Inputs.ToolResult_9.Data_1             :=  TO_UINT(_word);         // IW244
            _word.%B0 := _data_in[15];
            _word.%B1 := _data_in[14];
            Inputs.ToolResult_9.Data_2             :=  TO_UINT(_word);         // IW246
            _word.%B0 := _data_in[17];
            _word.%B1 := _data_in[16];
            Inputs.ToolResult_9.Data_3             :=  TO_UINT(_word);         // IW248
                                                                                    // IW250
            //***************************************************************

            //*************************ToolResult_10*************************
            _retVal := Siemens.Simatic.DistributedIO.ReadData((Config.HWIDs.HwID_ToolResult_10) ,_data_in);
            IF _retVal > WORD#0 THEN
                Messenger.Activate(UINT#1615, eAxoMessageCategory#Error);
                Status.Error.Id := UINT#1615;
                RETURN;
            END_IF;

            _word.%B0 := _data_in[1];
            _word.%B1 := _data_in[0];
            Inputs.ToolResult_10.MatchingRate       :=  TO_UINT(_word);        // IW252
            _word.%B0 := _data_in[3];
            _word.%B1 := _data_in[2];
            Inputs.ToolResult_10.MatchingRateMAX    :=  TO_UINT(_word);        // IW254
            _word.%B0 := _data_in[5];
            _word.%B1 := _data_in[4];
            Inputs.ToolResult_10.MatchingRateMIN    :=  TO_UINT(_word);        // IW256
            _word.%B0 := _data_in[7];
            _word.%B1 := _data_in[6];
            Inputs.ToolResult_10.LowerThreshold     :=  TO_UINT(_word);        // IW258
            _word.%B0 := _data_in[9];
            _word.%B1 := _data_in[8];
            Inputs.ToolResult_10.UpperThreshold     :=  TO_UINT(_word);        // IW260
            _word.%B0 := _data_in[11];
            _word.%B1 := _data_in[10];
            Inputs.ToolResult_10.DecimalPointPosition:=  TO_UINT(_word);       // IW262
            _word.%B0 := _data_in[13];
            _word.%B1 := _data_in[12];
            Inputs.ToolResult_10.Data_1             :=  TO_UINT(_word);        // IW264
            _word.%B0 := _data_in[15];
            _word.%B1 := _data_in[14];
            Inputs.ToolResult_10.Data_2             :=  TO_UINT(_word);        // IW266
            _word.%B0 := _data_in[17];
            _word.%B1 := _data_in[16];
            Inputs.ToolResult_10.Data_3             :=  TO_UINT(_word);        // IW268
                                                                                    // IW270
            //***************************************************************

            //*************************ToolResult_11*************************
            _retVal := Siemens.Simatic.DistributedIO.ReadData((Config.HWIDs.HwID_ToolResult_11) ,_data_in);
            IF _retVal > WORD#0 THEN
                Messenger.Activate(UINT#1616, eAxoMessageCategory#Error);
                Status.Error.Id := UINT#1616;
                RETURN;
            END_IF;

            _word.%B0 := _data_in[1];
            _word.%B1 := _data_in[0];
            Inputs.ToolResult_11.MatchingRate       :=  TO_UINT(_word);        // IW272
            _word.%B0 := _data_in[3];
            _word.%B1 := _data_in[2];
            Inputs.ToolResult_11.MatchingRateMAX    :=  TO_UINT(_word);        // IW274
            _word.%B0 := _data_in[5];
            _word.%B1 := _data_in[4];
            Inputs.ToolResult_11.MatchingRateMIN    :=  TO_UINT(_word);        // IW276
            _word.%B0 := _data_in[7];
            _word.%B1 := _data_in[6];
            Inputs.ToolResult_11.LowerThreshold     :=  TO_UINT(_word);        // IW278
            _word.%B0 := _data_in[9];
            _word.%B1 := _data_in[8];
            Inputs.ToolResult_11.UpperThreshold     :=  TO_UINT(_word);        // IW280
            _word.%B0 := _data_in[11];
            _word.%B1 := _data_in[10];
            Inputs.ToolResult_11.DecimalPointPosition:=  TO_UINT(_word);       // IW282
            _word.%B0 := _data_in[13];
            _word.%B1 := _data_in[12];
            Inputs.ToolResult_11.Data_1             :=  TO_UINT(_word);        // IW284
            _word.%B0 := _data_in[15];
            _word.%B1 := _data_in[14];
            Inputs.ToolResult_11.Data_2             :=  TO_UINT(_word);        // IW286
            _word.%B0 := _data_in[17];
            _word.%B1 := _data_in[16];
            Inputs.ToolResult_11.Data_3             :=  TO_UINT(_word);        // IW288
                                                                                    // IW290
            //***************************************************************

            //*************************ToolResult_12*************************
            _retVal := Siemens.Simatic.DistributedIO.ReadData((Config.HWIDs.HwID_ToolResult_12) ,_data_in);
            IF _retVal > WORD#0 THEN
                Messenger.Activate(UINT#1617, eAxoMessageCategory#Error);
                Status.Error.Id := UINT#1617;
                RETURN;
            END_IF;

            _word.%B0 := _data_in[1];
            _word.%B1 := _data_in[0];
            Inputs.ToolResult_12.MatchingRate       :=  TO_UINT(_word);        // IW292
            _word.%B0 := _data_in[3];
            _word.%B1 := _data_in[2];
            Inputs.ToolResult_12.MatchingRateMAX    :=  TO_UINT(_word);        // IW294
            _word.%B0 := _data_in[5];
            _word.%B1 := _data_in[4];
            Inputs.ToolResult_12.MatchingRateMIN    :=  TO_UINT(_word);        // IW296
            _word.%B0 := _data_in[7];
            _word.%B1 := _data_in[6];
            Inputs.ToolResult_12.LowerThreshold     :=  TO_UINT(_word);        // IW298
            _word.%B0 := _data_in[9];
            _word.%B1 := _data_in[8];
            Inputs.ToolResult_12.UpperThreshold     :=  TO_UINT(_word);        // IW300
            _word.%B0 := _data_in[11];
            _word.%B1 := _data_in[10];
            Inputs.ToolResult_12.DecimalPointPosition:=  TO_UINT(_word);       // IW302
            _word.%B0 := _data_in[13];
            _word.%B1 := _data_in[12];
            Inputs.ToolResult_12.Data_1             :=  TO_UINT(_word);        // IW304
            _word.%B0 := _data_in[15];
            _word.%B1 := _data_in[14];
            Inputs.ToolResult_12.Data_2             :=  TO_UINT(_word);        // IW306
            _word.%B0 := _data_in[17];
            _word.%B1 := _data_in[16];
            Inputs.ToolResult_12.Data_3             :=  TO_UINT(_word);        // IW308
                                                                                    // IW310
            //***************************************************************

            //*************************ToolResult_13*************************
            _retVal := Siemens.Simatic.DistributedIO.ReadData((Config.HWIDs.HwID_ToolResult_13) ,_data_in);
            IF _retVal > WORD#0 THEN
                Messenger.Activate(UINT#1618, eAxoMessageCategory#Error);
                Status.Error.Id := UINT#1618;
                RETURN;
            END_IF;

            _word.%B0 := _data_in[1];
            _word.%B1 := _data_in[0];
            Inputs.ToolResult_13.MatchingRate       :=  TO_UINT(_word);        // IW312
            _word.%B0 := _data_in[3];
            _word.%B1 := _data_in[2];
            Inputs.ToolResult_13.MatchingRateMAX    :=  TO_UINT(_word);        // IW314
            _word.%B0 := _data_in[5];
            _word.%B1 := _data_in[4];
            Inputs.ToolResult_13.MatchingRateMIN    :=  TO_UINT(_word);        // IW316
            _word.%B0 := _data_in[7];
            _word.%B1 := _data_in[6];
            Inputs.ToolResult_13.LowerThreshold     :=  TO_UINT(_word);        // IW318
            _word.%B0 := _data_in[9];
            _word.%B1 := _data_in[8];
            Inputs.ToolResult_13.UpperThreshold     :=  TO_UINT(_word);        // IW320
            _word.%B0 := _data_in[11];
            _word.%B1 := _data_in[10];
            Inputs.ToolResult_13.DecimalPointPosition:=  TO_UINT(_word);       // IW322
            _word.%B0 := _data_in[13];
            _word.%B1 := _data_in[12];
            Inputs.ToolResult_13.Data_1             :=  TO_UINT(_word);        // IW324
            _word.%B0 := _data_in[15];
            _word.%B1 := _data_in[14];
            Inputs.ToolResult_13.Data_2             :=  TO_UINT(_word);        // IW326
            _word.%B0 := _data_in[17];
            _word.%B1 := _data_in[16];
            Inputs.ToolResult_13.Data_3             :=  TO_UINT(_word);        // IW328
                                                                                    // IW330
            //***************************************************************

            //*************************ToolResult_14*************************
            _retVal := Siemens.Simatic.DistributedIO.ReadData((Config.HWIDs.HwID_ToolResult_14) ,_data_in);
            IF _retVal > WORD#0 THEN
                Messenger.Activate(UINT#1619, eAxoMessageCategory#Error);
                Status.Error.Id := UINT#1619;
                RETURN;
            END_IF;

            _word.%B0 := _data_in[1];
            _word.%B1 := _data_in[0];
            Inputs.ToolResult_14.MatchingRate       :=  TO_UINT(_word);        // IW332
            _word.%B0 := _data_in[3];
            _word.%B1 := _data_in[2];
            Inputs.ToolResult_14.MatchingRateMAX    :=  TO_UINT(_word);        // IW334
            _word.%B0 := _data_in[5];
            _word.%B1 := _data_in[4];
            Inputs.ToolResult_14.MatchingRateMIN    :=  TO_UINT(_word);        // IW336
            _word.%B0 := _data_in[7];
            _word.%B1 := _data_in[6];
            Inputs.ToolResult_14.LowerThreshold     :=  TO_UINT(_word);        // IW338
            _word.%B0 := _data_in[9];
            _word.%B1 := _data_in[8];
            Inputs.ToolResult_14.UpperThreshold     :=  TO_UINT(_word);        // IW340
            _word.%B0 := _data_in[11];
            _word.%B1 := _data_in[10];
            Inputs.ToolResult_14.DecimalPointPosition:=  TO_UINT(_word);       // IW342
            _word.%B0 := _data_in[13];
            _word.%B1 := _data_in[12];
            Inputs.ToolResult_14.Data_1             :=  TO_UINT(_word);        // IW344
            _word.%B0 := _data_in[15];
            _word.%B1 := _data_in[14];
            Inputs.ToolResult_14.Data_2             :=  TO_UINT(_word);        // IW346
            _word.%B0 := _data_in[17];
            _word.%B1 := _data_in[16];
            Inputs.ToolResult_14.Data_3             :=  TO_UINT(_word);        // IW348
                                                                                    // IW350
            //***************************************************************

            //*************************ToolResult_15*************************
            _retVal := Siemens.Simatic.DistributedIO.ReadData((Config.HWIDs.HwID_ToolResult_15) ,_data_in);
            IF _retVal > WORD#0 THEN
                Messenger.Activate(UINT#1620, eAxoMessageCategory#Error);
                Status.Error.Id := UINT#1620;
                RETURN;
            END_IF;

            _word.%B0 := _data_in[1];
            _word.%B1 := _data_in[0];
            Inputs.ToolResult_15.MatchingRate       :=  TO_UINT(_word);        // IW352
            _word.%B0 := _data_in[3];
            _word.%B1 := _data_in[2];
            Inputs.ToolResult_15.MatchingRateMAX    :=  TO_UINT(_word);        // IW354
            _word.%B0 := _data_in[5];
            _word.%B1 := _data_in[4];
            Inputs.ToolResult_15.MatchingRateMIN    :=  TO_UINT(_word);        // IW356
            _word.%B0 := _data_in[7];
            _word.%B1 := _data_in[6];
            Inputs.ToolResult_15.LowerThreshold     :=  TO_UINT(_word);        // IW358
            _word.%B0 := _data_in[9];
            _word.%B1 := _data_in[8];
            Inputs.ToolResult_15.UpperThreshold     :=  TO_UINT(_word);        // IW360
            _word.%B0 := _data_in[11];
            _word.%B1 := _data_in[10];
            Inputs.ToolResult_15.DecimalPointPosition:=  TO_UINT(_word);       // IW362
            _word.%B0 := _data_in[13];
            _word.%B1 := _data_in[12];
            Inputs.ToolResult_15.Data_1             :=  TO_UINT(_word);        // IW364
            _word.%B0 := _data_in[15];
            _word.%B1 := _data_in[14];
            Inputs.ToolResult_15.Data_2             :=  TO_UINT(_word);        // IW366
            _word.%B0 := _data_in[17];
            _word.%B1 := _data_in[16];
            Inputs.ToolResult_15.Data_3             :=  TO_UINT(_word);        // IW368
                                                                                    // IW370
            //***************************************************************

            //*************************ToolResult_16*************************
            _retVal := Siemens.Simatic.DistributedIO.ReadData((Config.HWIDs.HwID_ToolResult_16) ,_data_in);
            IF _retVal > WORD#0 THEN
                Messenger.Activate(UINT#1621, eAxoMessageCategory#Error);
                Status.Error.Id := UINT#1621;
                RETURN;
            END_IF;

            _word.%B0 := _data_in[1];
            _word.%B1 := _data_in[0];
            Inputs.ToolResult_16.MatchingRate       :=  TO_UINT(_word);        // IW372
            _word.%B0 := _data_in[3];
            _word.%B1 := _data_in[2];
            Inputs.ToolResult_16.MatchingRateMAX    :=  TO_UINT(_word);        // IW374
            _word.%B0 := _data_in[5];
            _word.%B1 := _data_in[4];
            Inputs.ToolResult_16.MatchingRateMIN    :=  TO_UINT(_word);        // IW376
            _word.%B0 := _data_in[7];
            _word.%B1 := _data_in[6];
            Inputs.ToolResult_16.LowerThreshold     :=  TO_UINT(_word);        // IW378
            _word.%B0 := _data_in[9];
            _word.%B1 := _data_in[8];
            Inputs.ToolResult_16.UpperThreshold     :=  TO_UINT(_word);        // IW380
            _word.%B0 := _data_in[11];
            _word.%B1 := _data_in[10];
            Inputs.ToolResult_16.DecimalPointPosition:=  TO_UINT(_word);       // IW382
            _word.%B0 := _data_in[13];
            _word.%B1 := _data_in[12];
            Inputs.ToolResult_16.Data_1             :=  TO_UINT(_word);        // IW384
            _word.%B0 := _data_in[15];
            _word.%B1 := _data_in[14];
            Inputs.ToolResult_16.Data_2             :=  TO_UINT(_word);        // IW386
            _word.%B0 := _data_in[17];
            _word.%B1 := _data_in[16];
            Inputs.ToolResult_16.Data_3             :=  TO_UINT(_word);        // IW388
                                                                                    // IW390
            //***************************************************************

            //*************************ToolResult_17*************************
            _retVal := Siemens.Simatic.DistributedIO.ReadData((Config.HWIDs.HwID_ToolResult_17) ,_data_in);
            IF _retVal > WORD#0 THEN
                Messenger.Activate(UINT#1622, eAxoMessageCategory#Error);
                Status.Error.Id := UINT#1622;
                RETURN;
            END_IF;

            _word.%B0 := _data_in[1];
            _word.%B1 := _data_in[0];
            Inputs.ToolResult_17.MatchingRate       :=  TO_UINT(_word);        // IW392
            _word.%B0 := _data_in[3];
            _word.%B1 := _data_in[2];
            Inputs.ToolResult_17.MatchingRateMAX    :=  TO_UINT(_word);        // IW394
            _word.%B0 := _data_in[5];
            _word.%B1 := _data_in[4];
            Inputs.ToolResult_17.MatchingRateMIN    :=  TO_UINT(_word);        // IW396
            _word.%B0 := _data_in[7];
            _word.%B1 := _data_in[6];
            Inputs.ToolResult_17.LowerThreshold     :=  TO_UINT(_word);        // IW398
            _word.%B0 := _data_in[9];
            _word.%B1 := _data_in[8];
            Inputs.ToolResult_17.UpperThreshold     :=  TO_UINT(_word);        // IW400
            _word.%B0 := _data_in[11];
            _word.%B1 := _data_in[10];
            Inputs.ToolResult_17.DecimalPointPosition:=  TO_UINT(_word);       // IW402
            _word.%B0 := _data_in[13];
            _word.%B1 := _data_in[12];
            Inputs.ToolResult_17.Data_1             :=  TO_UINT(_word);        // IW404
            _word.%B0 := _data_in[15];
            _word.%B1 := _data_in[14];
            Inputs.ToolResult_17.Data_2             :=  TO_UINT(_word);        // IW406
            _word.%B0 := _data_in[17];
            _word.%B1 := _data_in[16];
            Inputs.ToolResult_17.Data_3             :=  TO_UINT(_word);        // IW408
                                                                                    // IW410
            //***************************************************************

            //*************************ToolResult_18*************************
            _retVal := Siemens.Simatic.DistributedIO.ReadData((Config.HWIDs.HwID_ToolResult_18) ,_data_in);
            IF _retVal > WORD#0 THEN
                Messenger.Activate(UINT#1623, eAxoMessageCategory#Error);
                Status.Error.Id := UINT#1623;
                RETURN;
            END_IF;

            _word.%B0 := _data_in[1];
            _word.%B1 := _data_in[0];
            Inputs.ToolResult_18.MatchingRate       :=  TO_UINT(_word);        // IW412
            _word.%B0 := _data_in[3];
            _word.%B1 := _data_in[2];
            Inputs.ToolResult_18.MatchingRateMAX    :=  TO_UINT(_word);        // IW414
            _word.%B0 := _data_in[5];
            _word.%B1 := _data_in[4];
            Inputs.ToolResult_18.MatchingRateMIN    :=  TO_UINT(_word);        // IW416
            _word.%B0 := _data_in[7];
            _word.%B1 := _data_in[6];
            Inputs.ToolResult_18.LowerThreshold     :=  TO_UINT(_word);        // IW418
            _word.%B0 := _data_in[9];
            _word.%B1 := _data_in[8];
            Inputs.ToolResult_18.UpperThreshold     :=  TO_UINT(_word);        // IW420
            _word.%B0 := _data_in[11];
            _word.%B1 := _data_in[10];
            Inputs.ToolResult_18.DecimalPointPosition:=  TO_UINT(_word);       // IW422
            _word.%B0 := _data_in[13];
            _word.%B1 := _data_in[12];
            Inputs.ToolResult_18.Data_1             :=  TO_UINT(_word);        // IW424
            _word.%B0 := _data_in[15];
            _word.%B1 := _data_in[14];
            Inputs.ToolResult_18.Data_2             :=  TO_UINT(_word);        // IW426
            _word.%B0 := _data_in[17];
            _word.%B1 := _data_in[16];
            Inputs.ToolResult_18.Data_3             :=  TO_UINT(_word);        // IW428
                                                                                    // IW430
            //***************************************************************

            //*************************ToolResult_19*************************
            _retVal := Siemens.Simatic.DistributedIO.ReadData((Config.HWIDs.HwID_ToolResult_19) ,_data_in);
            IF _retVal > WORD#0 THEN
                Messenger.Activate(UINT#1624, eAxoMessageCategory#Error);
                Status.Error.Id := UINT#1624;
                RETURN;
            END_IF;

            _word.%B0 := _data_in[1];
            _word.%B1 := _data_in[0];
            Inputs.ToolResult_19.MatchingRate       :=  TO_UINT(_word);        // IW432
            _word.%B0 := _data_in[3];
            _word.%B1 := _data_in[2];
            Inputs.ToolResult_19.MatchingRateMAX    :=  TO_UINT(_word);        // IW434
            _word.%B0 := _data_in[5];
            _word.%B1 := _data_in[4];
            Inputs.ToolResult_19.MatchingRateMIN    :=  TO_UINT(_word);        // IW436
            _word.%B0 := _data_in[7];
            _word.%B1 := _data_in[6];
            Inputs.ToolResult_19.LowerThreshold     :=  TO_UINT(_word);        // IW438
            _word.%B0 := _data_in[9];
            _word.%B1 := _data_in[8];
            Inputs.ToolResult_19.UpperThreshold     :=  TO_UINT(_word);        // IW440
            _word.%B0 := _data_in[11];
            _word.%B1 := _data_in[10];
            Inputs.ToolResult_19.DecimalPointPosition:=  TO_UINT(_word);       // IW442
            _word.%B0 := _data_in[13];
            _word.%B1 := _data_in[12];
            Inputs.ToolResult_19.Data_1             :=  TO_UINT(_word);        // IW444
            _word.%B0 := _data_in[15];
            _word.%B1 := _data_in[14];
            Inputs.ToolResult_19.Data_2             :=  TO_UINT(_word);        // IW446
            _word.%B0 := _data_in[17];
            _word.%B1 := _data_in[16];
            Inputs.ToolResult_19.Data_3             :=  TO_UINT(_word);        // IW448
                                                                                    // IW450
            //***************************************************************

            //*************************ToolResult_20*************************
            _retVal := Siemens.Simatic.DistributedIO.ReadData((Config.HWIDs.HwID_ToolResult_20) ,_data_in);
            IF _retVal > WORD#0 THEN
                Messenger.Activate(UINT#1625, eAxoMessageCategory#Error);
                Status.Error.Id := UINT#1625;
                RETURN;
            END_IF;

            _word.%B0 := _data_in[1];
            _word.%B1 := _data_in[0];
            Inputs.ToolResult_20.MatchingRate       :=  TO_UINT(_word);        // IW452
            _word.%B0 := _data_in[3];
            _word.%B1 := _data_in[2];
            Inputs.ToolResult_20.MatchingRateMAX    :=  TO_UINT(_word);        // IW454
            _word.%B0 := _data_in[5];
            _word.%B1 := _data_in[4];
            Inputs.ToolResult_20.MatchingRateMIN    :=  TO_UINT(_word);        // IW456
            _word.%B0 := _data_in[7];
            _word.%B1 := _data_in[6];
            Inputs.ToolResult_20.LowerThreshold     :=  TO_UINT(_word);        // IW458
            _word.%B0 := _data_in[9];
            _word.%B1 := _data_in[8];
            Inputs.ToolResult_20.UpperThreshold     :=  TO_UINT(_word);        // IW460
            _word.%B0 := _data_in[11];
            _word.%B1 := _data_in[10];
            Inputs.ToolResult_20.DecimalPointPosition:=  TO_UINT(_word);       // IW462
            _word.%B0 := _data_in[13];
            _word.%B1 := _data_in[12];
            Inputs.ToolResult_20.Data_1             :=  TO_UINT(_word);        // IW464
            _word.%B0 := _data_in[15];
            _word.%B1 := _data_in[14];
            Inputs.ToolResult_20.Data_2             :=  TO_UINT(_word);        // IW466
            _word.%B0 := _data_in[17];
            _word.%B1 := _data_in[16];
            Inputs.ToolResult_20.Data_3             :=  TO_UINT(_word);        // IW468
                                                                                    // IW470
            //***************************************************************

            //*************************ToolResult_21*************************
            _retVal := Siemens.Simatic.DistributedIO.ReadData((Config.HWIDs.HwID_ToolResult_21) ,_data_in);
            IF _retVal > WORD#0 THEN
                Messenger.Activate(UINT#1626, eAxoMessageCategory#Error);
                Status.Error.Id := UINT#1626;
                RETURN;
            END_IF;

            _word.%B0 := _data_in[1];
            _word.%B1 := _data_in[0];
            Inputs.ToolResult_21.MatchingRate       :=  TO_UINT(_word);        // IW472
            _word.%B0 := _data_in[3];
            _word.%B1 := _data_in[2];
            Inputs.ToolResult_21.MatchingRateMAX    :=  TO_UINT(_word);        // IW474
            _word.%B0 := _data_in[5];
            _word.%B1 := _data_in[4];
            Inputs.ToolResult_21.MatchingRateMIN    :=  TO_UINT(_word);        // IW476
            _word.%B0 := _data_in[7];
            _word.%B1 := _data_in[6];
            Inputs.ToolResult_21.LowerThreshold     :=  TO_UINT(_word);        // IW478
            _word.%B0 := _data_in[9];
            _word.%B1 := _data_in[8];
            Inputs.ToolResult_21.UpperThreshold     :=  TO_UINT(_word);        // IW480
            _word.%B0 := _data_in[11];
            _word.%B1 := _data_in[10];
            Inputs.ToolResult_21.DecimalPointPosition:=  TO_UINT(_word);       // IW482
            _word.%B0 := _data_in[13];
            _word.%B1 := _data_in[12];
            Inputs.ToolResult_21.Data_1             :=  TO_UINT(_word);        // IW484
            _word.%B0 := _data_in[15];
            _word.%B1 := _data_in[14];
            Inputs.ToolResult_21.Data_2             :=  TO_UINT(_word);        // IW486
            _word.%B0 := _data_in[17];
            _word.%B1 := _data_in[16];
            Inputs.ToolResult_21.Data_3             :=  TO_UINT(_word);        // IW488
                                                                                    // IW490
            //***************************************************************

            //*************************ToolResult_22*************************
            _retVal := Siemens.Simatic.DistributedIO.ReadData((Config.HWIDs.HwID_ToolResult_22) ,_data_in);
            IF _retVal > WORD#0 THEN
                Messenger.Activate(UINT#1627, eAxoMessageCategory#Error);
                Status.Error.Id := UINT#1627;
                RETURN;
            END_IF;

            _word.%B0 := _data_in[1];
            _word.%B1 := _data_in[0];
            Inputs.ToolResult_22.MatchingRate       :=  TO_UINT(_word);        // IW492
            _word.%B0 := _data_in[3];
            _word.%B1 := _data_in[2];
            Inputs.ToolResult_22.MatchingRateMAX    :=  TO_UINT(_word);        // IW494
            _word.%B0 := _data_in[5];
            _word.%B1 := _data_in[4];
            Inputs.ToolResult_22.MatchingRateMIN    :=  TO_UINT(_word);        // IW496
            _word.%B0 := _data_in[7];
            _word.%B1 := _data_in[6];
            Inputs.ToolResult_22.LowerThreshold     :=  TO_UINT(_word);        // IW498
            _word.%B0 := _data_in[9];
            _word.%B1 := _data_in[8];
            Inputs.ToolResult_22.UpperThreshold     :=  TO_UINT(_word);        // IW500
            _word.%B0 := _data_in[11];
            _word.%B1 := _data_in[10];
            Inputs.ToolResult_22.DecimalPointPosition:=  TO_UINT(_word);       // IW502
            _word.%B0 := _data_in[13];
            _word.%B1 := _data_in[12];
            Inputs.ToolResult_22.Data_1             :=  TO_UINT(_word);        // IW504
            _word.%B0 := _data_in[15];
            _word.%B1 := _data_in[14];
            Inputs.ToolResult_22.Data_2             :=  TO_UINT(_word);        // IW506
            _word.%B0 := _data_in[17];
            _word.%B1 := _data_in[16];
            Inputs.ToolResult_22.Data_3             :=  TO_UINT(_word);        // IW508
                                                                                    // IW510
            //***************************************************************

            //*************************ToolResult_23*************************
            _retVal := Siemens.Simatic.DistributedIO.ReadData((Config.HWIDs.HwID_ToolResult_23) ,_data_in);
            IF _retVal > WORD#0 THEN
                Messenger.Activate(UINT#1628, eAxoMessageCategory#Error);
                Status.Error.Id := UINT#1628;
                RETURN;
            END_IF;

            _word.%B0 := _data_in[1];
            _word.%B1 := _data_in[0];
            Inputs.ToolResult_23.MatchingRate       :=  TO_UINT(_word);        // IW512
            _word.%B0 := _data_in[3];
            _word.%B1 := _data_in[2];
            Inputs.ToolResult_23.MatchingRateMAX    :=  TO_UINT(_word);        // IW514
            _word.%B0 := _data_in[5];
            _word.%B1 := _data_in[4];
            Inputs.ToolResult_23.MatchingRateMIN    :=  TO_UINT(_word);        // IW516
            _word.%B0 := _data_in[7];
            _word.%B1 := _data_in[6];
            Inputs.ToolResult_23.LowerThreshold     :=  TO_UINT(_word);        // IW518
            _word.%B0 := _data_in[9];
            _word.%B1 := _data_in[8];
            Inputs.ToolResult_23.UpperThreshold     :=  TO_UINT(_word);        // IW520
            _word.%B0 := _data_in[11];
            _word.%B1 := _data_in[10];
            Inputs.ToolResult_23.DecimalPointPosition:=  TO_UINT(_word);       // IW522
            _word.%B0 := _data_in[13];
            _word.%B1 := _data_in[12];
            Inputs.ToolResult_23.Data_1             :=  TO_UINT(_word);        // IW524
            _word.%B0 := _data_in[15];
            _word.%B1 := _data_in[14];
            Inputs.ToolResult_23.Data_2             :=  TO_UINT(_word);        // IW526
            _word.%B0 := _data_in[17];
            _word.%B1 := _data_in[16];
            Inputs.ToolResult_23.Data_3             :=  TO_UINT(_word);        // IW528
                                                                                    // IW530
            //***************************************************************

            //*************************ToolResult_24*************************
            _retVal := Siemens.Simatic.DistributedIO.ReadData((Config.HWIDs.HwID_ToolResult_24) ,_data_in);
            IF _retVal > WORD#0 THEN
                Messenger.Activate(UINT#1629, eAxoMessageCategory#Error);
                Status.Error.Id := UINT#1629;
                RETURN;
            END_IF;

            _word.%B0 := _data_in[1];
            _word.%B1 := _data_in[0];
            Inputs.ToolResult_24.MatchingRate       :=  TO_UINT(_word);        // IW532
            _word.%B0 := _data_in[3];
            _word.%B1 := _data_in[2];
            Inputs.ToolResult_24.MatchingRateMAX    :=  TO_UINT(_word);        // IW534
            _word.%B0 := _data_in[5];
            _word.%B1 := _data_in[4];
            Inputs.ToolResult_24.MatchingRateMIN    :=  TO_UINT(_word);        // IW536
            _word.%B0 := _data_in[7];
            _word.%B1 := _data_in[6];
            Inputs.ToolResult_24.LowerThreshold     :=  TO_UINT(_word);        // IW538
            _word.%B0 := _data_in[9];
            _word.%B1 := _data_in[8];
            Inputs.ToolResult_24.UpperThreshold     :=  TO_UINT(_word);        // IW540
            _word.%B0 := _data_in[11];
            _word.%B1 := _data_in[10];
            Inputs.ToolResult_24.DecimalPointPosition:=  TO_UINT(_word);       // IW542
            _word.%B0 := _data_in[13];
            _word.%B1 := _data_in[12];
            Inputs.ToolResult_24.Data_1             :=  TO_UINT(_word);        // IW544
            _word.%B0 := _data_in[15];
            _word.%B1 := _data_in[14];
            Inputs.ToolResult_24.Data_2             :=  TO_UINT(_word);        // IW546
            _word.%B0 := _data_in[17];
            _word.%B1 := _data_in[16];
            Inputs.ToolResult_24.Data_3             :=  TO_UINT(_word);        // IW548
                                                                                    // IW550
            //***************************************************************

            //*************************ToolResult_25*************************
            _retVal := Siemens.Simatic.DistributedIO.ReadData((Config.HWIDs.HwID_ToolResult_25) ,_data_in);
            IF _retVal > WORD#0 THEN
                Messenger.Activate(UINT#1630, eAxoMessageCategory#Error);
                Status.Error.Id := UINT#1630;
                RETURN;
            END_IF;

            _word.%B0 := _data_in[1];
            _word.%B1 := _data_in[0];
            Inputs.ToolResult_25.MatchingRate       :=  TO_UINT(_word);        // IW552
            _word.%B0 := _data_in[3];
            _word.%B1 := _data_in[2];
            Inputs.ToolResult_25.MatchingRateMAX    :=  TO_UINT(_word);        // IW554
            _word.%B0 := _data_in[5];
            _word.%B1 := _data_in[4];
            Inputs.ToolResult_25.MatchingRateMIN    :=  TO_UINT(_word);        // IW556
            _word.%B0 := _data_in[7];
            _word.%B1 := _data_in[6];
            Inputs.ToolResult_25.LowerThreshold     :=  TO_UINT(_word);        // IW558
            _word.%B0 := _data_in[9];
            _word.%B1 := _data_in[8];
            Inputs.ToolResult_25.UpperThreshold     :=  TO_UINT(_word);        // IW560
            _word.%B0 := _data_in[11];
            _word.%B1 := _data_in[10];
            Inputs.ToolResult_25.DecimalPointPosition:=  TO_UINT(_word);       // IW562
            _word.%B0 := _data_in[13];
            _word.%B1 := _data_in[12];
            Inputs.ToolResult_25.Data_1             :=  TO_UINT(_word);        // IW564
            _word.%B0 := _data_in[15];
            _word.%B1 := _data_in[14];
            Inputs.ToolResult_25.Data_2             :=  TO_UINT(_word);        // IW566
            _word.%B0 := _data_in[17];
            _word.%B1 := _data_in[16];
            Inputs.ToolResult_25.Data_3             :=  TO_UINT(_word);        // IW568
                                                                                    // IW570
            //***************************************************************

            //*************************ToolResult_26*************************
            _retVal := Siemens.Simatic.DistributedIO.ReadData((Config.HWIDs.HwID_ToolResult_26) ,_data_in);
            IF _retVal > WORD#0 THEN
                Messenger.Activate(UINT#1631, eAxoMessageCategory#Error);
                Status.Error.Id := UINT#1631;
                RETURN;
            END_IF;

            _word.%B0 := _data_in[1];
            _word.%B1 := _data_in[0];
            Inputs.ToolResult_26.MatchingRate       :=  TO_UINT(_word);        // IW572
            _word.%B0 := _data_in[3];
            _word.%B1 := _data_in[2];
            Inputs.ToolResult_26.MatchingRateMAX    :=  TO_UINT(_word);        // IW574
            _word.%B0 := _data_in[5];
            _word.%B1 := _data_in[4];
            Inputs.ToolResult_26.MatchingRateMIN    :=  TO_UINT(_word);        // IW576
            _word.%B0 := _data_in[7];
            _word.%B1 := _data_in[6];
            Inputs.ToolResult_26.LowerThreshold     :=  TO_UINT(_word);        // IW578
            _word.%B0 := _data_in[9];
            _word.%B1 := _data_in[8];
            Inputs.ToolResult_26.UpperThreshold     :=  TO_UINT(_word);        // IW580
            _word.%B0 := _data_in[11];
            _word.%B1 := _data_in[10];
            Inputs.ToolResult_26.DecimalPointPosition:=  TO_UINT(_word);       // IW582
            _word.%B0 := _data_in[13];
            _word.%B1 := _data_in[12];
            Inputs.ToolResult_26.Data_1             :=  TO_UINT(_word);        // IW584
            _word.%B0 := _data_in[15];
            _word.%B1 := _data_in[14];
            Inputs.ToolResult_26.Data_2             :=  TO_UINT(_word);        // IW586
            _word.%B0 := _data_in[17];
            _word.%B1 := _data_in[16];
            Inputs.ToolResult_26.Data_3             :=  TO_UINT(_word);        // IW588
                                                                                    // IW590
            //***************************************************************

            //*************************ToolResult_27*************************
            _retVal := Siemens.Simatic.DistributedIO.ReadData((Config.HWIDs.HwID_ToolResult_27) ,_data_in);
            IF _retVal > WORD#0 THEN
                Messenger.Activate(UINT#1632, eAxoMessageCategory#Error);
                Status.Error.Id := UINT#1632;
                RETURN;
            END_IF;

            _word.%B0 := _data_in[1];
            _word.%B1 := _data_in[0];
            Inputs.ToolResult_27.MatchingRate       :=  TO_UINT(_word);        // IW592
            _word.%B0 := _data_in[3];
            _word.%B1 := _data_in[2];
            Inputs.ToolResult_27.MatchingRateMAX    :=  TO_UINT(_word);        // IW594
            _word.%B0 := _data_in[5];
            _word.%B1 := _data_in[4];
            Inputs.ToolResult_27.MatchingRateMIN    :=  TO_UINT(_word);        // IW596
            _word.%B0 := _data_in[7];
            _word.%B1 := _data_in[6];
            Inputs.ToolResult_27.LowerThreshold     :=  TO_UINT(_word);        // IW598
            _word.%B0 := _data_in[9];
            _word.%B1 := _data_in[8];
            Inputs.ToolResult_27.UpperThreshold     :=  TO_UINT(_word);        // IW600
            _word.%B0 := _data_in[11];
            _word.%B1 := _data_in[10];
            Inputs.ToolResult_27.DecimalPointPosition:=  TO_UINT(_word);       // IW602
            _word.%B0 := _data_in[13];
            _word.%B1 := _data_in[12];
            Inputs.ToolResult_27.Data_1             :=  TO_UINT(_word);        // IW604
            _word.%B0 := _data_in[15];
            _word.%B1 := _data_in[14];
            Inputs.ToolResult_27.Data_2             :=  TO_UINT(_word);        // IW606
            _word.%B0 := _data_in[17];
            _word.%B1 := _data_in[16];
            Inputs.ToolResult_27.Data_3             :=  TO_UINT(_word);        // IW608
                                                                                    // IW610
            //***************************************************************

            //*************************ToolResult_28*************************
            _retVal := Siemens.Simatic.DistributedIO.ReadData((Config.HWIDs.HwID_ToolResult_28) ,_data_in);
            IF _retVal > WORD#0 THEN
                Messenger.Activate(UINT#1633, eAxoMessageCategory#Error);
                Status.Error.Id := UINT#1633;
                RETURN;
            END_IF;

            _word.%B0 := _data_in[1];
            _word.%B1 := _data_in[0];
            Inputs.ToolResult_28.MatchingRate       :=  TO_UINT(_word);        // IW612
            _word.%B0 := _data_in[3];
            _word.%B1 := _data_in[2];
            Inputs.ToolResult_28.MatchingRateMAX    :=  TO_UINT(_word);        // IW614
            _word.%B0 := _data_in[5];
            _word.%B1 := _data_in[4];
            Inputs.ToolResult_28.MatchingRateMIN    :=  TO_UINT(_word);        // IW616
            _word.%B0 := _data_in[7];
            _word.%B1 := _data_in[6];
            Inputs.ToolResult_28.LowerThreshold     :=  TO_UINT(_word);        // IW618
            _word.%B0 := _data_in[9];
            _word.%B1 := _data_in[8];
            Inputs.ToolResult_28.UpperThreshold     :=  TO_UINT(_word);        // IW620
            _word.%B0 := _data_in[11];
            _word.%B1 := _data_in[10];
            Inputs.ToolResult_28.DecimalPointPosition:=  TO_UINT(_word);       // IW622
            _word.%B0 := _data_in[13];
            _word.%B1 := _data_in[12];
            Inputs.ToolResult_28.Data_1             :=  TO_UINT(_word);        // IW624
            _word.%B0 := _data_in[15];
            _word.%B1 := _data_in[14];
            Inputs.ToolResult_28.Data_2             :=  TO_UINT(_word);        // IW626
            _word.%B0 := _data_in[17];
            _word.%B1 := _data_in[16];
            Inputs.ToolResult_28.Data_3             :=  TO_UINT(_word);        // IW628
                                                                                    // IW630
            //***************************************************************

            //*************************ToolResult_29*************************
            _retVal := Siemens.Simatic.DistributedIO.ReadData((Config.HWIDs.HwID_ToolResult_29) ,_data_in);
            IF _retVal > WORD#0 THEN
                Messenger.Activate(UINT#1634, eAxoMessageCategory#Error);
                Status.Error.Id := UINT#1634;
                RETURN;
            END_IF;

            _word.%B0 := _data_in[1];
            _word.%B1 := _data_in[0];
            Inputs.ToolResult_29.MatchingRate       :=  TO_UINT(_word);        // IW632
            _word.%B0 := _data_in[3];
            _word.%B1 := _data_in[2];
            Inputs.ToolResult_29.MatchingRateMAX    :=  TO_UINT(_word);        // IW634
            _word.%B0 := _data_in[5];
            _word.%B1 := _data_in[4];
            Inputs.ToolResult_29.MatchingRateMIN    :=  TO_UINT(_word);        // IW636
            _word.%B0 := _data_in[7];
            _word.%B1 := _data_in[6];
            Inputs.ToolResult_29.LowerThreshold     :=  TO_UINT(_word);        // IW638
            _word.%B0 := _data_in[9];
            _word.%B1 := _data_in[8];
            Inputs.ToolResult_29.UpperThreshold     :=  TO_UINT(_word);        // IW640
            _word.%B0 := _data_in[11];
            _word.%B1 := _data_in[10];
            Inputs.ToolResult_29.DecimalPointPosition:=  TO_UINT(_word);       // IW642
            _word.%B0 := _data_in[13];
            _word.%B1 := _data_in[12];
            Inputs.ToolResult_29.Data_1             :=  TO_UINT(_word);        // IW644
            _word.%B0 := _data_in[15];
            _word.%B1 := _data_in[14];
            Inputs.ToolResult_29.Data_2             :=  TO_UINT(_word);        // IW646
            _word.%B0 := _data_in[17];
            _word.%B1 := _data_in[16];
            Inputs.ToolResult_29.Data_3             :=  TO_UINT(_word);        // IW648
                                                                                    // IW650
            //***************************************************************

            //*************************ToolResult_30*************************
            _retVal := Siemens.Simatic.DistributedIO.ReadData((Config.HWIDs.HwID_ToolResult_30) ,_data_in);
            IF _retVal > WORD#0 THEN
                Messenger.Activate(UINT#1635, eAxoMessageCategory#Error);
                Status.Error.Id := UINT#1635;
                RETURN;
            END_IF;

            _word.%B0 := _data_in[1];
            _word.%B1 := _data_in[0];
            Inputs.ToolResult_30.MatchingRate       :=  TO_UINT(_word);        // IW652
            _word.%B0 := _data_in[3];
            _word.%B1 := _data_in[2];
            Inputs.ToolResult_30.MatchingRateMAX    :=  TO_UINT(_word);        // IW654
            _word.%B0 := _data_in[5];
            _word.%B1 := _data_in[4];
            Inputs.ToolResult_30.MatchingRateMIN    :=  TO_UINT(_word);        // IW656
            _word.%B0 := _data_in[7];
            _word.%B1 := _data_in[6];
            Inputs.ToolResult_30.LowerThreshold     :=  TO_UINT(_word);        // IW658
            _word.%B0 := _data_in[9];
            _word.%B1 := _data_in[8];
            Inputs.ToolResult_30.UpperThreshold     :=  TO_UINT(_word);        // IW660
            _word.%B0 := _data_in[11];
            _word.%B1 := _data_in[10];
            Inputs.ToolResult_30.DecimalPointPosition:=  TO_UINT(_word);       // IW662
            _word.%B0 := _data_in[13];
            _word.%B1 := _data_in[12];
            Inputs.ToolResult_30.Data_1             :=  TO_UINT(_word);        // IW664
            _word.%B0 := _data_in[15];
            _word.%B1 := _data_in[14];
            Inputs.ToolResult_30.Data_2             :=  TO_UINT(_word);        // IW666
            _word.%B0 := _data_in[17];
            _word.%B1 := _data_in[16];
            Inputs.ToolResult_30.Data_3             :=  TO_UINT(_word);        // IW668
                                                                                    // IW670
            //***************************************************************

            //*************************ToolResult_31*************************
            _retVal := Siemens.Simatic.DistributedIO.ReadData((Config.HWIDs.HwID_ToolResult_31) ,_data_in);
            IF _retVal > WORD#0 THEN
                Messenger.Activate(UINT#1636, eAxoMessageCategory#Error);
                Status.Error.Id := UINT#1636;
                RETURN;
            END_IF;

            _word.%B0 := _data_in[1];
            _word.%B1 := _data_in[0];
            Inputs.ToolResult_31.MatchingRate       :=  TO_UINT(_word);        // IW672
            _word.%B0 := _data_in[3];
            _word.%B1 := _data_in[2];
            Inputs.ToolResult_31.MatchingRateMAX    :=  TO_UINT(_word);        // IW674
            _word.%B0 := _data_in[5];
            _word.%B1 := _data_in[4];
            Inputs.ToolResult_31.MatchingRateMIN    :=  TO_UINT(_word);        // IW676
            _word.%B0 := _data_in[7];
            _word.%B1 := _data_in[6];
            Inputs.ToolResult_31.LowerThreshold     :=  TO_UINT(_word);        // IW678
            _word.%B0 := _data_in[9];
            _word.%B1 := _data_in[8];
            Inputs.ToolResult_31.UpperThreshold     :=  TO_UINT(_word);        // IW680
            _word.%B0 := _data_in[11];
            _word.%B1 := _data_in[10];
            Inputs.ToolResult_31.DecimalPointPosition:=  TO_UINT(_word);       // IW682
            _word.%B0 := _data_in[13];
            _word.%B1 := _data_in[12];
            Inputs.ToolResult_31.Data_1             :=  TO_UINT(_word);        // IW684
            _word.%B0 := _data_in[15];
            _word.%B1 := _data_in[14];
            Inputs.ToolResult_31.Data_2             :=  TO_UINT(_word);        // IW686
            _word.%B0 := _data_in[17];
            _word.%B1 := _data_in[16];
            Inputs.ToolResult_31.Data_3             :=  TO_UINT(_word);        // IW688
                                                                                    // IW690
            //***************************************************************

            //*************************ToolResult_32*************************
            _retVal := Siemens.Simatic.DistributedIO.ReadData((Config.HWIDs.HwID_ToolResult_32) ,_data_in);
            IF _retVal > WORD#0 THEN
                Messenger.Activate(UINT#1637, eAxoMessageCategory#Error);
                Status.Error.Id := UINT#1637;
                RETURN;
            END_IF;

            _word.%B0 := _data_in[1];
            _word.%B1 := _data_in[0];
            Inputs.ToolResult_32.MatchingRate       :=  TO_UINT(_word);        // IW692
            _word.%B0 := _data_in[3];
            _word.%B1 := _data_in[2];
            Inputs.ToolResult_32.MatchingRateMAX    :=  TO_UINT(_word);        // IW694
            _word.%B0 := _data_in[5];
            _word.%B1 := _data_in[4];
            Inputs.ToolResult_32.MatchingRateMIN    :=  TO_UINT(_word);        // IW696
            _word.%B0 := _data_in[7];
            _word.%B1 := _data_in[6];
            Inputs.ToolResult_32.LowerThreshold     :=  TO_UINT(_word);        // IW698
            _word.%B0 := _data_in[9];
            _word.%B1 := _data_in[8];
            Inputs.ToolResult_32.UpperThreshold     :=  TO_UINT(_word);        // IW700
            _word.%B0 := _data_in[11];
            _word.%B1 := _data_in[10];
            Inputs.ToolResult_32.DecimalPointPosition:=  TO_UINT(_word);       // IW702
            _word.%B0 := _data_in[13];
            _word.%B1 := _data_in[12];
            Inputs.ToolResult_32.Data_1             :=  TO_UINT(_word);        // IW704
            _word.%B0 := _data_in[15];
            _word.%B1 := _data_in[14];
            Inputs.ToolResult_32.Data_2             :=  TO_UINT(_word);        // IW706
            _word.%B0 := _data_in[17];
            _word.%B1 := _data_in[16];
            Inputs.ToolResult_32.Data_3             :=  TO_UINT(_word);        // IW708
                                                                                    // IW710
            //***************************************************************
